// TIA Portal V21 export
FUNCTION_BLOCK "AoFb"   // FB106, LAD
{ S7_Optimized_Access := 'TRUE' }
// stored: AutoNumber false, MemoryReserve 100, SetENOAutomatically false
   VAR_INPUT
      AlwaysTrue : Bool;
      AlwaysFalse : Bool;
   END_VAR
   VAR
      Ao01 { S7_SetPoint := 'True'} : "AnalogOutputScaling";   // Mm01Ref
      Ao02 { S7_SetPoint := 'True'} : "AnalogOutputScaling";   // Cp01Ref
      Ao03 { S7_SetPoint := 'True'} : "AnalogOutputScaling";   // Cv01
      Ao04 { S7_SetPoint := 'True'} : "AnalogOutputScaling";   // AoSpare1
      Ao05 { S7_SetPoint := 'True'} : "AnalogOutputScaling";   // AoSpare2
      Ao06 { S7_SetPoint := 'True'} : "AnalogOutputScaling";   // AoSpare3
      Ao07 { S7_SetPoint := 'True'} : "AnalogOutputScaling";   // AoSpare4
      Ao08 { S7_SetPoint := 'True'} : "AnalogOutputScaling";   // AoSpare5
   END_VAR
BEGIN

REGION Network 2: Mm01Ref
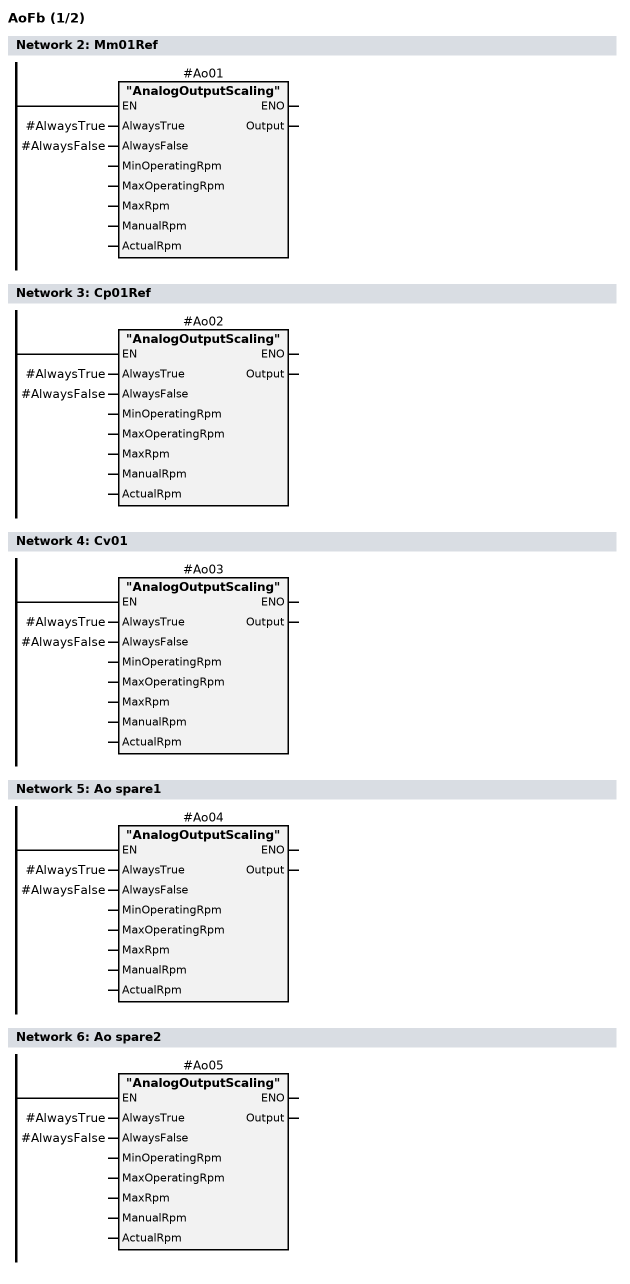
   RUNG wire#powerrail
      #Ao01(AlwaysTrue := #AlwaysTrue, AlwaysFalse := #AlwaysFalse, MinOperatingRpm :=, MaxOperatingRpm :=, MaxRpm :=, ManualRpm :=, ActualRpm :=, Output =>)
   END_RUNG
   // the same network as SCL:
   #Ao01(AlwaysTrue := #AlwaysTrue, AlwaysFalse := #AlwaysFalse);   // "AnalogOutputScaling"
END_REGION

REGION Network 3: Cp01Ref
   RUNG wire#powerrail
      #Ao02(AlwaysTrue := #AlwaysTrue, AlwaysFalse := #AlwaysFalse, MinOperatingRpm :=, MaxOperatingRpm :=, MaxRpm :=, ManualRpm :=, ActualRpm :=, Output =>)
   END_RUNG
   // the same network as SCL:
   #Ao02(AlwaysTrue := #AlwaysTrue, AlwaysFalse := #AlwaysFalse);   // "AnalogOutputScaling"
END_REGION

REGION Network 4: Cv01
   RUNG wire#powerrail
      #Ao03(AlwaysTrue := #AlwaysTrue, AlwaysFalse := #AlwaysFalse, MinOperatingRpm :=, MaxOperatingRpm :=, MaxRpm :=, ManualRpm :=, ActualRpm :=, Output =>)
   END_RUNG
   // the same network as SCL:
   #Ao03(AlwaysTrue := #AlwaysTrue, AlwaysFalse := #AlwaysFalse);   // "AnalogOutputScaling"
END_REGION

REGION Network 5: Ao spare1
   RUNG wire#powerrail
      #Ao04(AlwaysTrue := #AlwaysTrue, AlwaysFalse := #AlwaysFalse, MinOperatingRpm :=, MaxOperatingRpm :=, MaxRpm :=, ManualRpm :=, ActualRpm :=, Output =>)
   END_RUNG
   // the same network as SCL:
   #Ao04(AlwaysTrue := #AlwaysTrue, AlwaysFalse := #AlwaysFalse);   // "AnalogOutputScaling"
END_REGION

REGION Network 6: Ao spare2
   RUNG wire#powerrail
      #Ao05(AlwaysTrue := #AlwaysTrue, AlwaysFalse := #AlwaysFalse, MinOperatingRpm :=, MaxOperatingRpm :=, MaxRpm :=, ManualRpm :=, ActualRpm :=, Output =>)
   END_RUNG
   // the same network as SCL:
   #Ao05(AlwaysTrue := #AlwaysTrue, AlwaysFalse := #AlwaysFalse);   // "AnalogOutputScaling"
END_REGION

REGION Network 7: Ao spare3
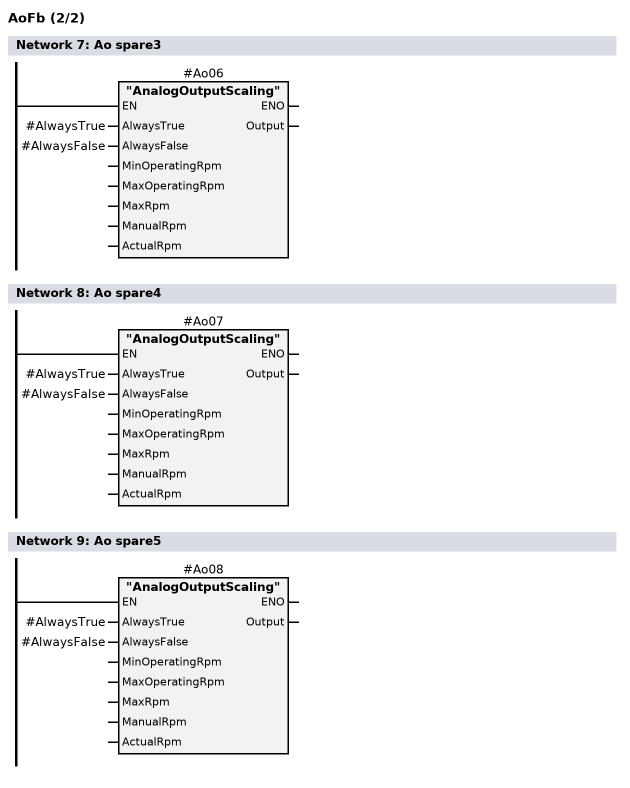
   RUNG wire#powerrail
      #Ao06(AlwaysTrue := #AlwaysTrue, AlwaysFalse := #AlwaysFalse, MinOperatingRpm :=, MaxOperatingRpm :=, MaxRpm :=, ManualRpm :=, ActualRpm :=, Output =>)
   END_RUNG
   // the same network as SCL:
   #Ao06(AlwaysTrue := #AlwaysTrue, AlwaysFalse := #AlwaysFalse);   // "AnalogOutputScaling"
END_REGION

REGION Network 8: Ao spare4
   RUNG wire#powerrail
      #Ao07(AlwaysTrue := #AlwaysTrue, AlwaysFalse := #AlwaysFalse, MinOperatingRpm :=, MaxOperatingRpm :=, MaxRpm :=, ManualRpm :=, ActualRpm :=, Output =>)
   END_RUNG
   // the same network as SCL:
   #Ao07(AlwaysTrue := #AlwaysTrue, AlwaysFalse := #AlwaysFalse);   // "AnalogOutputScaling"
END_REGION

REGION Network 9: Ao spare5
   RUNG wire#powerrail
      #Ao08(AlwaysTrue := #AlwaysTrue, AlwaysFalse := #AlwaysFalse, MinOperatingRpm :=, MaxOperatingRpm :=, MaxRpm :=, ManualRpm :=, ActualRpm :=, Output =>)
   END_RUNG
   // the same network as SCL:
   #Ao08(AlwaysTrue := #AlwaysTrue, AlwaysFalse := #AlwaysFalse);   // "AnalogOutputScaling"
END_REGION
END_FUNCTION_BLOCK
